// Mitsubishi GX Works2 project: double_Core   PLC: Q03UDV

PROGRAM MAIN
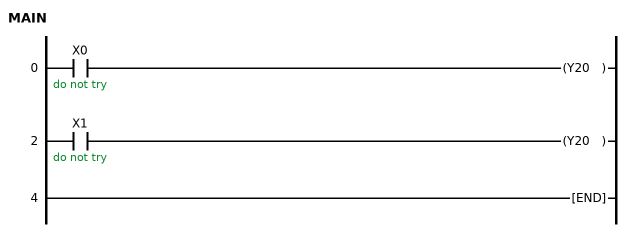
0     LD      X0  ; do not try
      OUT     Y20
2     LD      X1  ; do not try
      OUT     Y20
4     END
END_PROGRAM
